TYPE T_EXT_STRING : STRING(PARAM.MAX_EXT_STRING_LENGTH); END_TYPE

(* stored: Version 1.1.0.1, ProductVersion 3.1.4024.3
   DUT T_EXT_STRING: Id {1616d471-751d-4144-95c2-dce6a3fb50ed} *)
